(* IEC 61131-3 sources: BnR-JSONer/JSONer_exported/V1.0.1, 4 files *)

(* ---- JSON_Deserialize.st ---- *)
FUNCTION JSON_deserialize
	pActStr := pIn;
	freeBuffer := sizeIn;
	//================================================
	//Ignore first name member
	IF pUserVarName <> 0 THEN
		xStatus := findCharOrEnd(cIn := jsonAsciiColon, pStart := pActStr, maxLen := freeBuffer);
		IF xStatus > findError_OK THEN
			JSON_deserialize := JSONer_InputError;
			RETURN;
		END_IF;
		firstMemberArray := TRUE;
	END_IF;
	//================================================
	//Do Magic
	WHILE TRUE DO
		eStatus := JSON_var_deserialize(pFullVarName := pVarName, isArray := firstMemberArray, pStart := pActStr, size := freeBuffer);
		IF eStatus = JSONer_End THEN
			JSON_deserialize := JSONer_Ok;
			RETURN;
		ELSIF eStatus <> JSONer_Ok THEN
			JSON_deserialize := eStatus;
			RETURN;
		END_IF;
		firstMemberArray := FALSE;
	END_WHILE;
	//================================================
	JSON_deserialize := JSONer_Ok;
END_FUNCTION

FUNCTION JSON_var_deserialize
	//================================================
	// Copy basic var name
	brsmemset(ADR(varFullName),0, SIZEOF(varFullName));
	pFullNameNxtAddr := ADR(varFullName);
	pFullNameNxtAddr := brsstrcpy(pFullNameNxtAddr, pFullVarName);
	//================================================
	// Find var name - not used, if it's array -> for redirecting var types
	IF NOT isArray THEN
		xTempLen := findQuoation(pStart := pStart, maxLen := size);//Find start of name - by "
		IF xTempLen > findError_OK THEN
			JSON_var_deserialize := JSONer_End;
			RETURN;
		END_IF;
		pNameStart := pStart;
		xNameLen := findQuoation(pStart := pStart, maxLen := size);//Find end of name by "
		IF xNameLen > 32 THEN //findError_OK - Name can't be longer than 32 characters
			JSON_var_deserialize := JSONer_InputError;
			RETURN;
		END_IF;
		brsmemset(ADR(varName),0, SIZEOF(varName));
		brsmemcpy(ADR(varName), pNameStart, xNameLen);
		pFullNameNxtAddr := brsstrcpy(pFullNameNxtAddr, ADR('.'));
		pFullNameNxtAddr := brsstrcpy(pFullNameNxtAddr, ADR(varName));
	END_IF;
	//================================================
	//Find variable info in PVs
	xStatus := PV_ninfo(pv_name := ADR(varFullName), data_typ_p := ADR(varType), data_len_p := ADR(varLength), dimension_p := ADR(varDimension));
	IF xStatus <> 0 THEN
		JSON_var_deserialize := JSONer_VarNotFound;
		RETURN;
	END_IF;
	xStatus := PV_xgetadr(ADR(varFullName), ADR(varAddr), ADR(varSize));
	IF xStatus <> 0 THEN
		JSON_var_deserialize := JSONer_Error;
		RETURN;
	END_IF;
	//================================================
	//Extract value and decode

	IF varType = SYSLIB_IEC_TYPE_USER_DEFINED THEN //Structure
		// Remove {
		xTempLen := findChar(cIn := jsonAsciiLB, pStart := pStart, maxLen := size);
		IF xTempLen > findError_OK THEN
			JSON_var_deserialize := JSONer_InputError;
			RETURN;
		END_IF;
		// Find all variables inside
		FOR i := 0 TO (varDimension - 1) BY 1 DO
			eStatus := JSON_var_deserialize(pFullVarName := ADR(varFullName), isArray := FALSE, pStart := pStart, size := size);
			IF eStatus = JSONer_End OR eStatus = JSONer_VarNotFound THEN
				EXIT;
			ELSIF eStatus <> JSONer_Ok THEN
				JSON_var_deserialize := eStatus;
				RETURN;
			END_IF;
		END_FOR;

	ELSIF varType = SYSLIB_IEC_TYPE_USER_DEFINED_2 OR varDimension > 1 THEN //Array
		FOR i := 0 TO (varDimension - 1) BY 1 DO
			pVarFullNameExt := ADR(varFullNameExt);
			pVarFullNameExt := brsstrcpy(pVarFullNameExt, ADR(varFullName));
			pVarFullNameExt := brsstrcpy(pVarFullNameExt, ADR('['));
			varJsonStr := UDINT_TO_STRING(i);
			pVarFullNameExt := brsstrcpy(pVarFullNameExt, ADR(varJsonStr));
			pVarFullNameExt := brsstrcpy(pVarFullNameExt, ADR(']'));
			eStatus := JSON_var_deserialize(pFullVarName := ADR(varFullNameExt), isArray := TRUE, pStart := pStart, size := size);
			IF eStatus = JSONer_End OR eStatus = JSONer_VarNotFound THEN
				EXIT;
			ELSIF eStatus <> JSONer_Ok THEN
				JSON_var_deserialize := eStatus;
				RETURN;
			END_IF;
		END_FOR;

	ELSIF varType = SYSLIB_IEC_TYPE_BOOL THEN
		xTempLen := extractBool(pStart := pStart, maxLen := size, out := allTypes.tBool);
		IF xTempLen > findError_OK THEN
			JSON_var_deserialize := JSONer_InputError;
			RETURN;
		END_IF;
		brsmemcpy(varAddr, ADR(allTypes.tBool), varSize);

	ELSIF varType = SYSLIB_IEC_TYPE_SINT THEN
		xTempLen := findNumeric(pStart := pStart, maxLen := size);
		IF xTempLen > findError_OK THEN
			JSON_var_deserialize := JSONer_InputError;
			RETURN;
		END_IF;
		pValueStart := pStart;
		xTempLen := findNumericEnd(pStart := pStart, maxLen := size);
		IF (xTempLen + 1) > SIZEOF(varJsonStr) THEN
			JSON_var_deserialize := JSONer_InputError;
			RETURN;
		END_IF;
		brsmemset(ADR(varJsonStr),0, SIZEOF(varJsonStr));
		brsmemcpy(ADR(varJsonStr), pValueStart, xTempLen);
		allTypes.tSint := STRING_TO_SINT(varJsonStr);
		brsmemcpy(varAddr, ADR(allTypes.tSint), varSize);

	ELSIF varType = SYSLIB_IEC_TYPE_INT THEN
		xTempLen := findNumeric(pStart := pStart, maxLen := size);
		IF xTempLen > findError_OK THEN
			JSON_var_deserialize := JSONer_InputError;
			RETURN;
		END_IF;
		pValueStart := pStart;
		xTempLen := findNumericEnd(pStart := pStart, maxLen := size);
		IF (xTempLen + 1) > SIZEOF(varJsonStr) THEN
			JSON_var_deserialize := JSONer_InputError;
			RETURN;
		END_IF;
		brsmemset(ADR(varJsonStr),0, SIZEOF(varJsonStr));
		brsmemcpy(ADR(varJsonStr), pValueStart, xTempLen);
		allTypes.tInt := STRING_TO_INT(varJsonStr);
		brsmemcpy(varAddr, ADR(allTypes.tInt), varSize);

	ELSIF varType = SYSLIB_IEC_TYPE_DINT THEN
		xTempLen := findNumeric(pStart := pStart, maxLen := size);
		IF xTempLen > findError_OK THEN
			JSON_var_deserialize := JSONer_InputError;
			RETURN;
		END_IF;
		pValueStart := pStart;
		xTempLen := findNumericEnd(pStart := pStart, maxLen := size);
		IF (xTempLen + 1) > SIZEOF(varJsonStr) THEN
			JSON_var_deserialize := JSONer_InputError;
			RETURN;
		END_IF;
		brsmemset(ADR(varJsonStr),0, SIZEOF(varJsonStr));
		brsmemcpy(ADR(varJsonStr), pValueStart, xTempLen);
		allTypes.tDint := STRING_TO_DINT(varJsonStr);
		brsmemcpy(varAddr, ADR(allTypes.tDint), varSize);

	ELSIF varType = SYSLIB_IEC_TYPE_USINT THEN
		xTempLen := findNumeric(pStart := pStart, maxLen := size);
		IF xTempLen > findError_OK THEN
			JSON_var_deserialize := JSONer_InputError;
			RETURN;
		END_IF;
		pValueStart := pStart;
		xTempLen := findNumericEnd(pStart := pStart, maxLen := size);
		IF (xTempLen + 1) > SIZEOF(varJsonStr) THEN
			JSON_var_deserialize := JSONer_InputError;
			RETURN;
		END_IF;
		brsmemset(ADR(varJsonStr),0, SIZEOF(varJsonStr));
		brsmemcpy(ADR(varJsonStr), pValueStart, xTempLen);
		allTypes.tUsint := STRING_TO_USINT(varJsonStr);
		brsmemcpy(varAddr, ADR(allTypes.tUsint), varSize);

	ELSIF varType = SYSLIB_IEC_TYPE_UINT THEN
		xTempLen := findNumeric(pStart := pStart, maxLen := size);
		IF xTempLen > findError_OK THEN
			JSON_var_deserialize := JSONer_InputError;
			RETURN;
		END_IF;
		pValueStart := pStart;
		xTempLen := findNumericEnd(pStart := pStart, maxLen := size);
		IF (xTempLen + 1) > SIZEOF(varJsonStr) THEN
			JSON_var_deserialize := JSONer_InputError;
			RETURN;
		END_IF;
		brsmemset(ADR(varJsonStr),0, SIZEOF(varJsonStr));
		brsmemcpy(ADR(varJsonStr), pValueStart, xTempLen);
		allTypes.tUint := STRING_TO_UINT(varJsonStr);
		brsmemcpy(varAddr, ADR(allTypes.tUint), varSize);

	ELSIF varType = SYSLIB_IEC_TYPE_UDINT THEN
		xTempLen := findNumeric(pStart := pStart, maxLen := size);
		IF xTempLen > findError_OK THEN
			JSON_var_deserialize := JSONer_InputError;
			RETURN;
		END_IF;
		pValueStart := pStart;
		xTempLen := findNumericEnd(pStart := pStart, maxLen := size);
		IF (xTempLen + 1) > SIZEOF(varJsonStr) THEN
			JSON_var_deserialize := JSONer_InputError;
			RETURN;
		END_IF;
		brsmemset(ADR(varJsonStr),0, SIZEOF(varJsonStr));
		brsmemcpy(ADR(varJsonStr), pValueStart, xTempLen);
		allTypes.tUdint := STRING_TO_UDINT(varJsonStr);
		brsmemcpy(varAddr, ADR(allTypes.tUdint), varSize);

	ELSIF varType = SYSLIB_IEC_TYPE_REAL THEN
		xTempLen := findNumeric(pStart := pStart, maxLen := size);
		IF xTempLen > findError_OK THEN
			JSON_var_deserialize := JSONer_InputError;
			RETURN;
		END_IF;
		pValueStart := pStart;
		xTempLen := findNumericEnd(pStart := pStart, maxLen := size);
		IF (xTempLen + 1) > SIZEOF(varJsonStr) THEN
			JSON_var_deserialize := JSONer_InputError;
			RETURN;
		END_IF;
		brsmemset(ADR(varJsonStr),0, SIZEOF(varJsonStr));
		brsmemcpy(ADR(varJsonStr), pValueStart, xTempLen);
		allTypes.tReal := STRING_TO_REAL(varJsonStr);
		brsmemcpy(varAddr, ADR(allTypes.tReal), varSize);

	ELSIF varType = SYSLIB_IEC_TYPE_STRING THEN
		xTempLen := findQuoation(pStart := pStart, maxLen := size);
		IF xTempLen > findError_OK THEN
			JSON_var_deserialize := JSONer_InputError;
			RETURN;
		END_IF;
		pValueStart := pStart;
		xTempLen := findQuoation(pStart := pStart, maxLen := size);
		IF (xTempLen + 1) > varSize THEN
			JSON_var_deserialize := JSONer_InputError;
			RETURN;
		END_IF;
		brsmemset(varAddr,0, varSize);
		brsmemcpy(varAddr, pValueStart, xTempLen);

	ELSIF varType = SYSLIB_IEC_TYPE_DATE_AND_TIME THEN
		xTempLen := findQuoation(pStart := pStart, maxLen := size);
		IF xTempLen > findError_OK THEN
			JSON_var_deserialize := JSONer_InputError;
			RETURN;
		END_IF;
		pValueStart := pStart;
		xTempLen := findQuoation(pStart := pStart, maxLen := size);
		IF (xTempLen + 1) > SIZEOF(varJsonStr) THEN
			JSON_var_deserialize := JSONer_InputError;
			RETURN;
		END_IF;
		brsmemset(ADR(varJsonStr),0, SIZEOF(varJsonStr));
		brsmemcpy(ADR(varJsonStr), pValueStart, xTempLen);
		allTypes.tDt := STRING_TO_DT(varJsonStr);
		brsmemcpy(varAddr, ADR(allTypes.tDt), varSize);

	ELSIF varType = SYSLIB_IEC_TYPE_TIME THEN
		xTempLen := findQuoation(pStart := pStart, maxLen := size);
		IF xTempLen > findError_OK THEN
			JSON_var_deserialize := JSONer_InputError;
			RETURN;
		END_IF;
		pValueStart := pStart;
		xTempLen := findQuoation(pStart := pStart, maxLen := size);
		IF (xTempLen + 1) > SIZEOF(varJsonStr) THEN
			JSON_var_deserialize := JSONer_InputError;
			RETURN;
		END_IF;
		brsmemset(ADR(varJsonStr),0, SIZEOF(varJsonStr));
		brsmemcpy(ADR(varJsonStr), pValueStart, xTempLen);
		allTypes.tTime := STRING_TO_TIME(varJsonStr);
		brsmemcpy(varAddr, ADR(allTypes.tTime), varSize);

	ELSIF varType = SYSLIB_IEC_TYPE_DATE THEN
		xTempLen := findQuoation(pStart := pStart, maxLen := size);
		IF xTempLen > findError_OK THEN
			JSON_var_deserialize := JSONer_InputError;
			RETURN;
		END_IF;
		pValueStart := pStart;
		xTempLen := findQuoation(pStart := pStart, maxLen := size);
		IF (xTempLen + 1) > SIZEOF(varJsonStr) THEN
			JSON_var_deserialize := JSONer_InputError;
			RETURN;
		END_IF;
		brsmemset(ADR(varJsonStr),0, SIZEOF(varJsonStr));
		brsmemcpy(ADR(varJsonStr), pValueStart, xTempLen);
		allTypes.tDate := STRING_TO_DATE(varJsonStr);
		brsmemcpy(varAddr, ADR(allTypes.tDate), varSize);

	ELSIF varType = SYSLIB_IEC_TYPE_LREAL THEN
		xTempLen := findNumeric(pStart := pStart, maxLen := size);
		IF xTempLen > findError_OK THEN
			JSON_var_deserialize := JSONer_InputError;
			RETURN;
		END_IF;
		pValueStart := pStart;
		xTempLen := findNumericEnd(pStart := pStart, maxLen := size);
		IF (xTempLen + 1) > SIZEOF(varJsonStr) THEN
			JSON_var_deserialize := JSONer_InputError;
			RETURN;
		END_IF;
		brsmemset(ADR(varJsonStr),0, SIZEOF(varJsonStr));
		brsmemcpy(ADR(varJsonStr), pValueStart, xTempLen);
		allTypes.tLreal := STRING_TO_LREAL(varJsonStr);
		brsmemcpy(varAddr, ADR(allTypes.tLreal), varSize);

	ELSIF varType = SYSLIB_IEC_TYPE_TIME_OF_DAY THEN
		xTempLen := findQuoation(pStart := pStart, maxLen := size);
		IF xTempLen > findError_OK THEN
			JSON_var_deserialize := JSONer_InputError;
			RETURN;
		END_IF;
		pValueStart := pStart;
		xTempLen := findQuoation(pStart := pStart, maxLen := size);
		IF (xTempLen + 1) > SIZEOF(varJsonStr) THEN
			JSON_var_deserialize := JSONer_InputError;
			RETURN;
		END_IF;
		brsmemset(ADR(varJsonStr),0, SIZEOF(varJsonStr));
		brsmemcpy(ADR(varJsonStr), pValueStart, xTempLen);
		allTypes.tTod := STRING_TO_TOD(varJsonStr);
		brsmemcpy(varAddr, ADR(allTypes.tTod), varSize);

	ELSIF varType = SYSLIB_IEC_TYPE_BYTE THEN
		xTempLen := findNumeric(pStart := pStart, maxLen := size);
		IF xTempLen > findError_OK THEN
			JSON_var_deserialize := JSONer_InputError;
			RETURN;
		END_IF;
		pValueStart := pStart;
		xTempLen := findNumericEnd(pStart := pStart, maxLen := size);
		IF (xTempLen + 1) > SIZEOF(varJsonStr) THEN
			JSON_var_deserialize := JSONer_InputError;
			RETURN;
		END_IF;
		brsmemset(ADR(varJsonStr),0, SIZEOF(varJsonStr));
		brsmemcpy(ADR(varJsonStr), pValueStart, xTempLen);
		allTypes.tByte := STRING_TO_BYTE(varJsonStr);
		brsmemcpy(varAddr, ADR(allTypes.tByte), varSize);

	ELSIF varType = SYSLIB_IEC_TYPE_WORD THEN
		xTempLen := findNumeric(pStart := pStart, maxLen := size);
		IF xTempLen > findError_OK THEN
			JSON_var_deserialize := JSONer_InputError;
			RETURN;
		END_IF;
		pValueStart := pStart;
		xTempLen := findNumericEnd(pStart := pStart, maxLen := size);
		IF (xTempLen + 1) > SIZEOF(varJsonStr) THEN
			JSON_var_deserialize := JSONer_InputError;
			RETURN;
		END_IF;
		brsmemset(ADR(varJsonStr),0, SIZEOF(varJsonStr));
		brsmemcpy(ADR(varJsonStr), pValueStart, xTempLen);
		allTypes.tWord := STRING_TO_WORD(varJsonStr);
		brsmemcpy(varAddr, ADR(allTypes.tWord), varSize);

	ELSIF varType = SYSLIB_IEC_TYPE_DWORD THEN
		xTempLen := findNumeric(pStart := pStart, maxLen := size);
		IF xTempLen > findError_OK THEN
			JSON_var_deserialize := JSONer_InputError;
			RETURN;
		END_IF;
		pValueStart := pStart;
		xTempLen := findNumericEnd(pStart := pStart, maxLen := size);
		IF (xTempLen + 1) > SIZEOF(varJsonStr) THEN
			JSON_var_deserialize := JSONer_InputError;
			RETURN;
		END_IF;
		brsmemset(ADR(varJsonStr),0, SIZEOF(varJsonStr));
		brsmemcpy(ADR(varJsonStr), pValueStart, xTempLen);
		allTypes.tDword := STRING_TO_DWORD(varJsonStr);
		brsmemcpy(varAddr, ADR(allTypes.tDword), varSize);

	ELSIF varType = SYSLIB_IEC_TYPE_WSTRING THEN

	ELSE
		JSON_var_deserialize := JSONer_BadVarType;
		RETURN;
	END_IF;

	//================================================
	// Check the end
	xTempLen := findCharOrEnd(cIn := jsonAsciiComma, pStart := pStart, maxLen := size);
	IF xTempLen = findError_EndExceed THEN
		JSON_var_deserialize := JSONer_End;
	ELSIF xTempLen > findError_OK THEN
		JSON_var_deserialize := JSONer_InputError;
		RETURN;
	END_IF;

	JSON_var_deserialize := JSONer_Ok;
END_FUNCTION

(* ---- JSON_Serialize.st ---- *)
FUNCTION JSON_serialize
	freeBuffer := sizeOut;
	brsmemset(pOut, 0, sizeOut);
	//================================================
	//Get variable name and info
	IF pVarName = 0 THEN
		JSON_serialize := JSONer_InputError;
		RETURN;
	END_IF;
	brsstrcpy(ADR(varName), pVarName);
	xStatus := PV_ninfo(pv_name := ADR(varName), data_typ_p := ADR(dataTyp), data_len_p := ADR(dataLen), dimension_p := ADR(dataDim));
	IF xStatus <> 0 THEN
		JSON_serialize := JSONer_VarNotFound;
		RETURN;
	END_IF;
	//================================================
	//Start frame
	bufferAdrNext := pOut;
	bufferAdrNext := brsstrcpy(bufferAdrNext, ADR('{'));
	freeBuffer := freeBuffer - 2;
	//================================================
	//Start serializing
	//listTyp.data_typ listTyp.dimension
	eStatus := JSON_var_serialize(pFullVarName := ADR(varName), pVarName := pUserVarName, varDimension := UINT_TO_UDINT(dataDim), varType := UDINT_TO_USINT(dataTyp), firstMember := TRUE, pBuffer := bufferAdrNext, freeBuffer := freeBuffer);
	IF eStatus <> JSONer_Ok THEN
		JSON_serialize := eStatus;
		RETURN;
	END_IF;
	//================================================
	//End frame
	IF freeBuffer > 2 THEN
		bufferAdrNext := brsstrcpy(bufferAdrNext, ADR(' }'));
		freeBuffer := freeBuffer - 2;
	ELSE
		JSON_serialize := JSONer_SmallBuffer;
		RETURN;
	END_IF;
	size := sizeOut - freeBuffer;
	JSON_serialize := JSONer_Ok;
END_FUNCTION

//0 for structures and 15 for array of structures

FUNCTION JSON_var_serialize
	JSON_var_serialize := JSONer_Ok;
	//================================================
	//Value name
	IF varType >= 0 AND varType <= 21 AND varType <> 10 AND varType <> 20 THEN
		IF NOT ((varType = 0 AND firstMember = TRUE)) THEN //Pokud není struktura samostatná pro výpis -  AND varDimension < 2
			xStrLen := 6 + brsstrlen(pVarName);
			IF freeBuffer > xStrLen THEN
				pBuffer := brsstrcpy(pBuffer, ADR(' "'));
				pBuffer := brsstrcpy(pBuffer, pVarName);
				pBuffer := brsstrcpy(pBuffer, ADR('" : '));
				freeBuffer := freeBuffer - xStrLen;
			ELSE
				JSON_var_serialize := JSONer_SmallBuffer;
				RETURN;
			END_IF;
		END_IF;
	ELSE
		JSON_var_serialize := JSONer_BadVarType;
		RETURN;
	END_IF;
	//================================================
	//Start array
	IF varDimension > 1 AND NOT (varType = 0) THEN
		actDim := varDimension;
		IF freeBuffer > 2 THEN
			pBuffer := brsstrcpy(pBuffer, ADR(' ['));
			freeBuffer := freeBuffer - 2;
		ELSE
			JSON_var_serialize := JSONer_SmallBuffer;
			RETURN;
		END_IF;
	ELSE
		actDim := 1;
	END_IF;
	//================================================
	//Value serialize
	WHILE actDim > 0 DO
		copyConvStr := FALSE;
		//================================================
		structStrAdr := ADR(structFullNameMember);
		structStrAdr := brsstrcpy(structStrAdr, pFullVarName);
		IF varDimension > 1 AND NOT (varType = 0) THEN
			structStrAdr := brsstrcpy(structStrAdr, ADR('['));
			structItemName := UDINT_TO_STRING(varDimension - actDim);
			structStrAdr := brsstrcpy(structStrAdr, ADR(structItemName));
			structStrAdr := brsstrcpy(structStrAdr, ADR(']'));
			firstMember := FALSE;//
		END_IF;
		//================================================
		xStatus := PV_xgetadr(ADR(structFullNameMember), ADR(structItemAdr), ADR(structItemAdrLen));
		IF xStatus <> 0 THEN
			JSON_var_serialize := JSONer_Error;
			RETURN;
		END_IF;
		//================================================
		useQuoation := FALSE;
		copyConvStr := FALSE;
		IF varType = SYSLIB_IEC_TYPE_USER_DEFINED OR varType = SYSLIB_IEC_TYPE_USER_DEFINED_2 THEN
			//================================================
			//Init Object
			IF NOT firstMember THEN
				IF freeBuffer > 2 THEN
					pBuffer := brsstrcpy(pBuffer, ADR(' {'));
					freeBuffer := freeBuffer - 2;
				ELSE
					JSON_var_serialize := JSONer_SmallBuffer;
					RETURN;
				END_IF;
			END_IF;
			//================================================
			//Call structure members
			//structStrAdr := ADR(structFullNameMember);
			//structStrAdr := brsstrcpy(structStrAdr, pFullVarName);
			structStrAdr := brsstrcpy(structStrAdr, ADR('.'));
			structActIndex := 0;
			WHILE TRUE DO
				xStatus := PV_item(pv_name := pFullVarName, index := structActIndex, ADR(structItemName));
				IF xStatus = 0 AND structActIndex < 100 THEN
					brsstrcpy(structStrAdr, ADR(structItemName));
					xStatus := PV_ninfo(pv_name := ADR(structFullNameMember), data_typ_p := ADR(structItemType), data_len_p := ADR(structItemLen), dimension_p := ADR(structItemDimension));
					IF xStatus <> 0 THEN
						JSON_var_serialize := JSONer_Error;
						RETURN;
					END_IF;
					IF structActIndex > 0 THEN
						IF freeBuffer > 2 THEN
							pBuffer := brsstrcpy(pBuffer, ADR(' ,'));
							freeBuffer := freeBuffer - 2;
						ELSE
							JSON_var_serialize := JSONer_SmallBuffer;
							RETURN;
						END_IF;
					END_IF;
					eStatus := JSON_var_serialize(pFullVarName := ADR(structFullNameMember), pVarName := ADR(structItemName), varDimension := structItemDimension, varType := UDINT_TO_USINT(structItemType), firstMember := FALSE, pBuffer := pBuffer, freeBuffer := freeBuffer);
					IF eStatus <> JSONer_Ok THEN
						JSON_var_serialize := eStatus;
						RETURN;
					END_IF;
				ELSE
					EXIT;
				END_IF;
				structActIndex := structActIndex + 1;
			END_WHILE;

			//================================================
			//End Object
			IF NOT firstMember THEN
				IF freeBuffer > 2 THEN
					pBuffer := brsstrcpy(pBuffer, ADR(' }'));
					freeBuffer := freeBuffer - 2;
				ELSE
					JSON_var_serialize := JSONer_SmallBuffer;
					RETURN;
				END_IF;
			END_IF;
			//================================================
		ELSIF varType = SYSLIB_IEC_TYPE_BOOL THEN
			brsmemcpy(ADR(allTypes.tBool), structItemAdr, structItemAdrLen);
			IF allTypes.tBool THEN
				brsstrcpy(ADR(strValConv), ADR('true'));
			ELSE
				brsstrcpy(ADR(strValConv), ADR('false'));
			END_IF;
			copyConvStr := TRUE;

		ELSIF varType = SYSLIB_IEC_TYPE_SINT THEN
			brsmemcpy(ADR(allTypes.tSint), structItemAdr, structItemAdrLen);
			strValConv := SINT_TO_STRING(allTypes.tSint);
			copyConvStr := TRUE;

		ELSIF varType = SYSLIB_IEC_TYPE_INT THEN
			brsmemcpy(ADR(allTypes.tInt), structItemAdr, structItemAdrLen);
			strValConv := INT_TO_STRING(allTypes.tInt);
			copyConvStr := TRUE;

		ELSIF varType = SYSLIB_IEC_TYPE_DINT THEN
			brsmemcpy(ADR(allTypes.tDint), structItemAdr, structItemAdrLen);
			strValConv := DINT_TO_STRING(allTypes.tDint);
			copyConvStr := TRUE;

		ELSIF varType = SYSLIB_IEC_TYPE_USINT THEN
			brsmemcpy(ADR(allTypes.tUsint), structItemAdr, structItemAdrLen);
			strValConv := USINT_TO_STRING(allTypes.tUsint);
			copyConvStr := TRUE;

		ELSIF varType = SYSLIB_IEC_TYPE_UINT THEN
			brsmemcpy(ADR(allTypes.tUint), structItemAdr, structItemAdrLen);
			strValConv := UINT_TO_STRING(allTypes.tUint);
			copyConvStr := TRUE;

		ELSIF varType = SYSLIB_IEC_TYPE_UDINT THEN
			brsmemcpy(ADR(allTypes.tUdint), structItemAdr, structItemAdrLen);
			strValConv := UDINT_TO_STRING(allTypes.tUdint);
			copyConvStr := TRUE;
			useQuoation := FALSE;

		ELSIF varType = SYSLIB_IEC_TYPE_REAL THEN
			brsmemcpy(ADR(allTypes.tReal), structItemAdr, structItemAdrLen);
			strValConv := REAL_TO_STRING(allTypes.tReal);
			copyConvStr := TRUE;

		ELSIF varType = SYSLIB_IEC_TYPE_STRING THEN//This is can be much bigger than internal variable
			xStrLen := 2 + brsstrlen(ADR(structItemAdr));
			IF freeBuffer > xStrLen THEN
				pBuffer := brsstrcpy(pBuffer, ADR('"'));
				pBuffer := brsstrcpy(pBuffer, structItemAdr);
				pBuffer := brsstrcpy(pBuffer, ADR('"'));
				freeBuffer := freeBuffer - xStrLen;
			ELSE
				JSON_var_serialize := JSONer_SmallBuffer;
				RETURN;
			END_IF;

		ELSIF varType = SYSLIB_IEC_TYPE_DATE_AND_TIME THEN
			brsmemcpy(ADR(allTypes.tDt), structItemAdr, structItemAdrLen);
			strValConv := DT_TO_STRING(allTypes.tDt);
			copyConvStr := TRUE;
			useQuoation := TRUE;

		ELSIF varType = SYSLIB_IEC_TYPE_TIME THEN
			brsmemcpy(ADR(allTypes.tTime), structItemAdr, structItemAdrLen);
			strValConv := TIME_TO_STRING(allTypes.tTime);
			copyConvStr := TRUE;
			useQuoation := TRUE;

		ELSIF varType = SYSLIB_IEC_TYPE_DATE THEN
			brsmemcpy(ADR(allTypes.tDate), structItemAdr, structItemAdrLen);
			strValConv := DATE_TO_STRING(allTypes.tDate);
			copyConvStr := TRUE;
			useQuoation := TRUE;

		ELSIF varType = SYSLIB_IEC_TYPE_LREAL THEN
			brsmemcpy(ADR(allTypes.tLreal), structItemAdr, structItemAdrLen);
			strValConv := LREAL_TO_STRING(allTypes.tLreal);
			copyConvStr := TRUE;

		ELSIF varType = SYSLIB_IEC_TYPE_TIME_OF_DAY THEN
			brsmemcpy(ADR(allTypes.tTod), structItemAdr, structItemAdrLen);
			strValConv := TOD_TO_STRING(allTypes.tTod);
			copyConvStr := TRUE;
			useQuoation := TRUE;

		ELSIF varType = SYSLIB_IEC_TYPE_BYTE THEN
			brsmemcpy(ADR(allTypes.tByte), structItemAdr, structItemAdrLen);
			strValConv := BYTE_TO_STRING(allTypes.tByte);
			copyConvStr := TRUE;

		ELSIF varType = SYSLIB_IEC_TYPE_WORD THEN
			brsmemcpy(ADR(allTypes.tWord), structItemAdr, structItemAdrLen);
			strValConv := WORD_TO_STRING(allTypes.tWord);
			copyConvStr := TRUE;

		ELSIF varType = SYSLIB_IEC_TYPE_DWORD THEN
			brsmemcpy(ADR(allTypes.tDword), structItemAdr, structItemAdrLen);
			strValConv := DWORD_TO_STRING(allTypes.tDword);
			copyConvStr := TRUE;

		ELSIF varType = SYSLIB_IEC_TYPE_WSTRING THEN

		ELSE
			JSON_var_serialize := JSONer_BadVarType;
			RETURN;
		END_IF;
		//================================================
		//Converted values copy
		IF copyConvStr THEN
			xStrLen := brsstrlen(ADR(strValConv)) + 2 * BOOL_TO_DINT(useQuoation);
			IF freeBuffer > xStrLen THEN
				IF useQuoation THEN
					pBuffer := brsstrcpy(pBuffer, ADR('"'));
				END_IF;
				pBuffer := brsstrcpy(pBuffer, ADR(strValConv));
				IF useQuoation THEN
					pBuffer := brsstrcpy(pBuffer, ADR('"'));
				END_IF;
				freeBuffer := freeBuffer - xStrLen;
			ELSE
				JSON_var_serialize := JSONer_SmallBuffer;
				RETURN;
			END_IF;
		END_IF;
		//================================================
		//Array handling
		actDim := actDim - 1;
		IF actDim > 0 THEN
			IF freeBuffer > 2 THEN
				pBuffer := brsstrcpy(pBuffer, ADR(' ,'));
				freeBuffer := freeBuffer - 2;
			ELSE
				JSON_var_serialize := JSONer_SmallBuffer;
				RETURN;
			END_IF;
		END_IF;
	END_WHILE;

	IF JSON_var_serialize <> JSONer_Ok THEN
		RETURN;
	END_IF;
	//================================================
	//End Array
	IF varDimension > 1 AND NOT (varType = 0) THEN
		IF freeBuffer > 2 THEN
			pBuffer := brsstrcpy(pBuffer, ADR(' ]'));
			freeBuffer := freeBuffer - 2;
		ELSE
			JSON_var_serialize := JSONer_SmallBuffer;
			RETURN;
		END_IF;
	END_IF;
	//================================================
	JSON_var_serialize := JSONer_Ok;
END_FUNCTION

(* ---- JSON_Support.st ---- *)
//================================================
//
FUNCTION findChar
	FOR i := 0 TO maxLen BY 1 DO
		c ACCESS (pStart + i);
		IF c = cIn THEN
			maxLen := maxLen - (i + 1);
			pStart := pStart + i + 1;
			findChar := i;
			RETURN;
		ELSIF c = jsonAsciiNULL THEN
			findChar := findError_GenericError;
			RETURN;
		END_IF;
	END_FOR;
	findChar := findError_NotFound;
END_FUNCTION

//================================================
//

FUNCTION findCharOrEnd
	FOR i := 0 TO maxLen BY 1 DO
		c ACCESS (pStart + i);
		IF c = cIn THEN
			maxLen := maxLen - (i + 1);
			pStart := pStart + i + 1;
			findCharOrEnd := i;
			RETURN;
		ELSIF c = jsonAsciiRB OR c = jsonAsciiRSB THEN
			maxLen := maxLen - (i + 1);
			pStart := pStart + i + 1;
			findCharOrEnd := findError_EndExceed;
			RETURN;
		ELSIF c = jsonAsciiNULL THEN
			findCharOrEnd := findError_GenericError;
			RETURN;
		END_IF;
	END_FOR;
	findCharOrEnd := findError_NotFound;
END_FUNCTION

//================================================
//
FUNCTION findQuoation
	FOR i := 0 TO maxLen BY 1 DO
		c ACCESS (pStart + i);
		IF c = jsonAsciiDQuot THEN
			c ACCESS (pStart + i - 1);//Check the char before for backslash - it's will be char in string
			IF (c <> jsonAsciiBackslash AND i > 0) OR i = 0 THEN
				maxLen := maxLen - (i + 1);
				pStart := pStart + i + 1;
				findQuoation := i;
				RETURN;
			END_IF;
		ELSIF c = jsonAsciiRB OR c = jsonAsciiRSB THEN
			maxLen := maxLen - (i + 1);
			pStart := pStart + i + 1;
			findQuoation := findError_EndExceed;
			RETURN;
		ELSIF c = jsonAsciiNULL THEN
			findQuoation := findError_GenericError;
			RETURN;
		END_IF;
	END_FOR;
	findQuoation := findError_NotFound;
END_FUNCTION

//================================================
//
FUNCTION findNumeric
	FOR i := 0 TO maxLen BY 1 DO
		c ACCESS (pStart + i);
		IF (c >= jsonAscii0 AND c <= jsonAscii9) OR c = jsonAsciiPlus OR c = jsonAsciiMinus  THEN
			maxLen := maxLen - i;
			pStart := pStart + i;
			findNumeric := i;
			RETURN;
		ELSIF c = jsonAsciiRB OR c = jsonAsciiRSB THEN
			maxLen := maxLen - (i + 1);
			pStart := pStart + i + 1;
			findNumeric := findError_EndExceed;
			RETURN;
		ELSIF c = jsonAsciiNULL THEN
			findNumeric := findError_GenericError;
			RETURN;
		END_IF;
	END_FOR;
	findNumeric := findError_NotFound;
END_FUNCTION

//================================================
//
FUNCTION findNumericEnd
	FOR i := 0 TO maxLen BY 1 DO
		c ACCESS (pStart + i);
		IF c = jsonAsciiLF OR c = jsonAsciiSP OR c = jsonAsciiTab OR c = jsonAsciiCR OR c = jsonAsciiComma THEN
			maxLen := maxLen - i;
			pStart := pStart + i;
			findNumericEnd := i;
			RETURN;
		ELSIF c = jsonAsciiRB OR c = jsonAsciiRSB THEN
			maxLen := maxLen - (i + 1);
			pStart := pStart + i + 1;
			findNumericEnd := findError_EndExceed;
			RETURN;
		ELSIF c = jsonAsciiNULL THEN
			findNumericEnd := findError_GenericError;
			RETURN;
		END_IF;
	END_FOR;
	findNumericEnd := findError_NotFound;
END_FUNCTION

//================================================
//
FUNCTION findWhitespace
	FOR i := 0 TO maxLen BY 1 DO
		c ACCESS (pStart + i);
		IF c = jsonAsciiLF OR c = jsonAsciiSP OR c = jsonAsciiTab OR c = jsonAsciiCR THEN
			maxLen := maxLen - i;
			pStart := pStart + i;
			findWhitespace := i;
			RETURN;
		ELSIF c = jsonAsciiRB OR c = jsonAsciiRSB THEN
			maxLen := maxLen - (i + 1);
			pStart := pStart + i + 1;
			findWhitespace := findError_EndExceed;
			RETURN;
		ELSIF c = jsonAsciiNULL THEN
			findWhitespace := findError_GenericError;
			RETURN;
		END_IF;
	END_FOR;
	findWhitespace := findError_NotFound;
END_FUNCTION

//================================================
//
FUNCTION extractBool
	il:= 0;
	FOR i := 0 TO maxLen BY 1 DO
		c ACCESS (pStart + i);
		IF c = jsonAscii0 THEN
			out := FALSE;
			EXIT;
		ELSIF c = jsonAscii1 THEN
			out := TRUE;
			EXIT;
		ELSIF c >= jsonAsciiSa AND c <= jsonAsciiSz THEN
			FOR il := 0 TO MIN(maxLen - i, SIZEOF(text)) BY 1 DO
				c ACCESS (pStart + i + il);
				IF c < jsonAsciiSa OR c > jsonAsciiSz THEN
					EXIT;
				END_IF;
			END_FOR;
			IF il > SIZEOF(text) THEN
				extractBool := findError_OutOfMem;
				RETURN;
			END_IF;
			brsmemset(ADR(text), 0, SIZEOF(text));
			brsmemcpy(ADR(text), pStart + i, il);
			IF brsstrcmp(ADR(text), ADR('true')) = 0 THEN
				out := TRUE;
			ELSIF brsstrcmp(ADR(text), ADR('false')) = 0 THEN
				out := FALSE;
			ELSE
				extractBool := findError_GenericError;
				RETURN;
			END_IF;
			EXIT;
		ELSIF c = jsonAsciiRB OR c = jsonAsciiRSB THEN
			extractBool := findError_EndExceed;
			RETURN;
		END_IF;
	END_FOR;
	IF i + il >= maxLen THEN
		extractBool := findError_OutOfMem;
	ELSE
		maxLen := maxLen - (i + il);
		pStart := pStart + i + il;
		extractBool := i + il;
	END_IF;
END_FUNCTION

(* ---- JSONer.fun ---- *)
(*Serialize*)

FUNCTION JSON_serialize : JSONer_Status_e (*JSON serializer*)
	VAR_INPUT
		pVarName : UDINT; (*Name of variable. In local variable use full path - [Program":"][Variable]...*)
		pUserVarName : UDINT := 0; (*User name if input variable are array and not struct*)
		pOut : UDINT; (*Outout buffer - String or USINT[]*)
		sizeOut : UDINT; (*Maximum size of buffer - SIZEOF(pOut)*)
	END_VAR
	VAR_IN_OUT
		size : UDINT; (*Outout used size in bytes*)
	END_VAR
	VAR
		freeBuffer : UDINT;
		bufferAdrNext : UDINT;
		xStatus : UINT;
		eStatus : JSONer_Status_e;
		dataTyp : UDINT;
		dataLen : UDINT;
		dataDim : UINT;
		varName : STRING[80];
	END_VAR
END_FUNCTION

FUNCTION JSON_var_serialize : JSONer_Status_e
	VAR_INPUT
		pFullVarName : UDINT;
		pVarName : UDINT := 0;
		varDimension : UDINT := 1;
		varType : USINT;
		firstMember : BOOL := FALSE;
	END_VAR
	VAR_IN_OUT
		pBuffer : UDINT;
		freeBuffer : UDINT;
	END_VAR
	VAR
		xStatus : UINT;
		eStatus : JSONer_Status_e;
		actDim : UDINT := 0;
		xStrLen : UDINT;
		allTypes : JSONer_types_t;
		strValConv : STRING[80];
		copyConvStr : BOOL;
		useQuoation : BOOL;
		structFullNameMember : STRING[254];
		structActIndex : UINT;
		structItemName : STRING[32];
		structStrAdr : UDINT;
		structItemType : UDINT;
		structItemLen : UDINT;
		structItemDimension : UINT;
		structItemAdr : UDINT;
		structItemAdrLen : UDINT;
	END_VAR
END_FUNCTION
(*Deserialize*)

FUNCTION JSON_deserialize : JSONer_Status_e (*JSON deserializer*)
	VAR_INPUT
		pVarName : UDINT; (*Name of variable. In local variable use full path - [Program":"][Variable]...*)
		pUserVarName : UDINT := 0; (*User variable name in JSON for array input - set to 0, if input variable is struct*)
		pIn : UDINT; (*JSON string input - pointer*)
		sizeIn : UDINT; (*Size of input string - for not overloop*)
	END_VAR
	VAR
		xStatus : UDINT;
		eStatus : JSONer_Status_e;
		pActStr : UDINT;
		freeBuffer : UDINT;
		firstMemberArray : BOOL := FALSE;
	END_VAR
END_FUNCTION

FUNCTION JSON_var_deserialize : JSONer_Status_e
	VAR_INPUT
		pFullVarName : UDINT;
		isArray : BOOL;
	END_VAR
	VAR_IN_OUT
		pStart : UDINT;
		size : UDINT;
	END_VAR
	VAR
		xStatus : UINT;
		eStatus : JSONer_Status_e;
		allTypes : JSONer_types_t;
		varName : STRING[34];
		varFullName : STRING[254];
		varFullNameExt : STRING[254];
		pVarFullNameExt : UDINT;
		xTempLen : UDINT;
		xNameLen : UDINT;
		pNameStart : UDINT;
		pFullNameNxtAddr : UDINT;
		varType : UDINT;
		varLength : UDINT;
		varDimension : UINT;
		varAddr : UDINT;
		varSize : UDINT;
		varJsonStr : STRING[30];
		pValueStart : UDINT;
		i : UDINT;
	END_VAR
END_FUNCTION
(*Supporting functions*)

FUNCTION extractBool : UDINT
	VAR_IN_OUT
		pStart : UDINT;
		maxLen : UDINT; (*Limit the finding lenght*)
		out : BOOL;
	END_VAR
	VAR
		i : UDINT := 0;
		il : UDINT := 0;
		c : REFERENCE TO USINT;
		text : STRING[10];
	END_VAR
END_FUNCTION

FUNCTION findChar : UDINT
	VAR_INPUT
		cIn : USINT;
	END_VAR
	VAR_IN_OUT
		pStart : UDINT;
		maxLen : UDINT; (*Limit the finding lenght*)
	END_VAR
	VAR
		i : UDINT;
		c : REFERENCE TO USINT;
	END_VAR
END_FUNCTION

FUNCTION findCharOrEnd : UDINT
	VAR_INPUT
		cIn : USINT;
	END_VAR
	VAR_IN_OUT
		pStart : UDINT;
		maxLen : UDINT; (*Limit the finding lenght*)
	END_VAR
	VAR
		i : UDINT;
		c : REFERENCE TO USINT;
	END_VAR
END_FUNCTION

FUNCTION findQuoation : UDINT
	VAR_IN_OUT
		pStart : UDINT;
		maxLen : UDINT; (*Limit the finding lenght*)
	END_VAR
	VAR
		i : UDINT;
		c : REFERENCE TO USINT;
	END_VAR
END_FUNCTION

FUNCTION findNumeric : UDINT
	VAR_IN_OUT
		pStart : UDINT;
		maxLen : UDINT; (*Limit the finding lenght*)
	END_VAR
	VAR
		i : UDINT;
		c : REFERENCE TO USINT;
	END_VAR
END_FUNCTION

FUNCTION findNumericEnd : UDINT
	VAR_IN_OUT
		pStart : UDINT;
		maxLen : UDINT; (*Limit the finding lenght*)
	END_VAR
	VAR
		i : UDINT;
		c : REFERENCE TO USINT;
	END_VAR
END_FUNCTION

FUNCTION findWhitespace : UDINT
	VAR_IN_OUT
		pStart : UDINT;
		maxLen : UDINT; (*Limit the finding lenght*)
	END_VAR
	VAR
		i : UDINT;
		c : REFERENCE TO USINT;
	END_VAR
END_FUNCTION
